{attribute 'qualified_only'}
{attribute 'strict'}
{attribute 'to_string'}
TYPE E_ErrorState :
(
	Healthy := 0, Warning:=1, Alarm:= 2, Disabled:=3
);
END_TYPE

(* stored: Version 1.1.0.1
   DUT E_ErrorState: Id {61fc1aa6-90b7-4efb-86f7-b3f659ed9d56} *)
